FUNCTION_BLOCK contadorTempoRestante (* Basic Function Block Type *)
  (* Standard: 61499-2 *)
  (* Version 0.0, 25/02/2026, Template *)
  PACKAGE Hidryco.HidrycoLib;
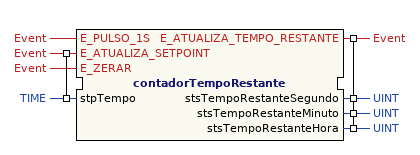
  EVENT_INPUT
    E_PULSO_1S;
    E_ATUALIZA_SETPOINT WITH stpTempo;
    E_ZERAR;
  END_EVENT
  EVENT_OUTPUT
    E_ATUALIZA_TEMPO_RESTANTE WITH stsTempoRestanteSegundo, stsTempoRestanteMinuto, stsTempoRestanteHora;
  END_EVENT
  VAR_INPUT
    stpTempo : TIME;
  END_VAR
  VAR_OUTPUT
    stsTempoRestanteSegundo : UINT;
    stsTempoRestanteMinuto : UINT;
    stsTempoRestanteHora : UINT;
  END_VAR
  VAR
    tempoAtual : UINT;
    tempoAtualSegundos : UINT;
    tempoAtualMinutos : UINT;
    tempoAtualHoras : UINT;
    totalSec : LINT;
    restanteSec : UDINT;
    rU : UDINT;
  END_VAR
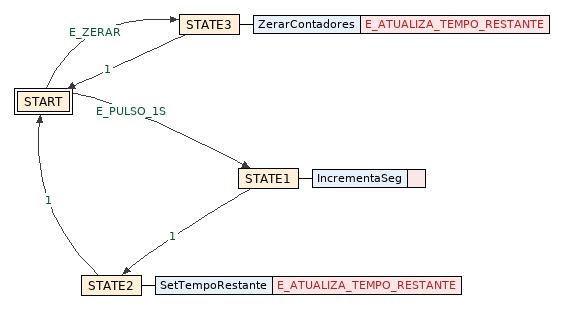
  EC_STATES
    START; (* Initial State *)
    STATE1 : IncrementaSeg;
    STATE2 : SetTempoRestante -> E_ATUALIZA_TEMPO_RESTANTE;
    STATE3 : ZerarContadores -> E_ATUALIZA_TEMPO_RESTANTE;
  END_STATES
  EC_TRANSITIONS
    START TO STATE1 := E_PULSO_1S;
    STATE1 TO STATE2 := 1;
    STATE2 TO START := 1;
    START TO STATE3 := E_ZERAR;
    STATE3 TO START := 1;
  END_TRANSITIONS
  ALGORITHM INIT IN ST: (* Initialization algorithm *)
;
  END_ALGORITHM
  ALGORITHM REQ IN ST: (* Normally executed algorithm *)
;
  END_ALGORITHM
  ALGORITHM IncrementaSeg IN ST:
tempoAtual := tempoAtual + 1;

tempoAtualHoras := tempoAtual / 3600;
tempoAtualMinutos := (tempoAtual MOD 3600) / 60;
tempoAtualSegundos := tempoAtual MOD 60;
;
  END_ALGORITHM
  ALGORITHM SetTempoRestante IN ST:
totalSec := TIME_TO_LINT(stpTempo) / 1000;

IF UINT_TO_UDINT(tempoAtual) >= LINT_TO_UDINT(totalSec) THEN
    restanteSec := 0;
ELSE
    restanteSec := LINT_TO_UDINT(totalSec) - tempoAtual;
END_IF;

stsTempoRestanteHora    := UDINT_TO_UINT(restanteSec / 3600);
stsTempoRestanteMinuto  := UDINT_TO_UINT((restanteSec MOD 3600) / 60);
stsTempoRestanteSegundo := UDINT_TO_UINT(restanteSec MOD 60);
  END_ALGORITHM
  ALGORITHM ZerarContadores IN ST:
tempoAtual := 0;
  END_ALGORITHM
END_FUNCTION_BLOCK
